TYPE ST_GantryXYZ_Config :
STRUCT
    CutterXOffsetX   : REAL;
    CutterXOffsetY   : REAL;
    CutterYOffsetX   : REAL;
    CutterYOffsetY   : REAL;
	CuttingSpeedXY	 :REAL;
    CuttingIdleTime  : REAL;
	GroovingSpeedXY  : REAL;
    GroovingSpeedZ   : REAL;
    GroovingIdleTime : REAL;
    RapidSpeedX      : REAL;
    RapidSpeedY      : REAL;
    RapidSpeedZ      : REAL;
    GlobalOffsetX    : REAL;
    GlobalOffsetY    : REAL;
	GlobalOffsetZ    : REAL; 
    RawBoardX        : REAL; 
    RawBoardY        : REAL;
	RawBoardZ        : REAL;
    SafeClearanceZ   : REAL; 
	AxisQ_SavedPos	 : LREAL;
END_STRUCT
END_TYPE

(* stored: Version 1.1.0.1, ProductVersion 3.1.4024.15
   DUT ST_GantryXYZ_Config: Id {9175d3d8-e623-4395-a625-175ecc53cdb9} *)
